FUNCTION_BLOCK fbVacuumPumpCtrl

VAR_INPUT
	IN_DevName:STRING;
	In_Enable:BOOL;
	In_Reset:BOOL;

	(*Starter Healthy Signal*)
	In_StarterOK:BOOL;

END_VAR

VAR_OUTPUT
	Out_MotorOn:BOOL;

END_VAR

VAR_IN_OUT
	MotorVar:structMotorDirect;	
	Station:structStationCtrl;
END_VAR


VAR

	MotorOn:BOOL;
	On_TOut: TON;
	On_TON: TON;
	Loc_OnPls: BOOL;
	OnPls: R_TRIG;
	Out_RSErr:BOOL;
	OnPosPls: F_TRIG;

END_VAR

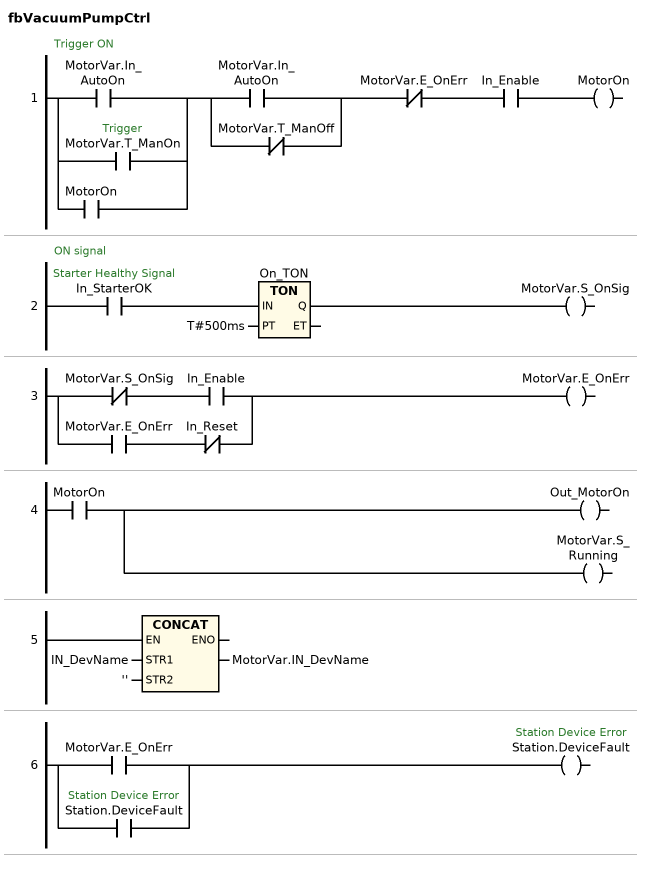
// NETWORK 1
// Trigger ON
//   MotorVar.T_ManOn: Trigger
MotorOn := (MotorVar.In_AutoOn OR MotorVar.T_ManOn OR MotorOn) AND (MotorVar.In_AutoOn OR NOT MotorVar.T_ManOff) AND NOT MotorVar.E_OnErr AND In_Enable;

// NETWORK 2
// ON signal
//   In_StarterOK: Starter Healthy Signal
On_TON(IN := In_StarterOK, PT := T#500ms); // TON
MotorVar.S_OnSig := On_TON.Q;

// NETWORK 3
MotorVar.E_OnErr := NOT MotorVar.S_OnSig AND In_Enable OR MotorVar.E_OnErr AND NOT In_Reset;

// NETWORK 4
Out_MotorOn := MotorOn;
MotorVar.S_Running := MotorOn;

// NETWORK 5
MotorVar.IN_DevName := CONCAT(STR1 := IN_DevName, STR2 := '');

// NETWORK 6
//   Station.DeviceFault: Station Device Error
Station.DeviceFault := MotorVar.E_OnErr OR Station.DeviceFault;

END_FUNCTION_BLOCK

(* stored: Version 1.1.0.1, ProductVersion 3.1.4018.2
   POU fbVacuumPumpCtrl: Id {0987a5af-fb3c-4b4e-8bc7-6256ee43ee2d}, SpecialFunc None *)
